DATA_BLOCK "DB_Parameters"
{ S7_Optimized_Access := 'TRUE' }
VERSION : 0.1
   VAR
      Level_Low : Real := 30.0;
      Level_High : Real := 80.0;
      Level_CritHigh : Real := 95.0;
      Source_Min : Real := 15.0;
      Source_Hyst_pct : Real := 5.0;
      Flow_Min : Real := 2.0;
      Flow_Validation : Time := T#10s;
      Restart_Delay : Time := T#30s;
      Run_Feedback_Timeout : Time := T#5s;
      Init_Delay : Time := T#2s;
      Maint_Test_Max : Time := T#60s;
      FreqStarts_Max : Int := 3;
      FreqStarts_Window_min : Int := 60;
      Current_Nominal : Real := 10.0;
      Current_High : Real := 12.0;
      Current_High_Delay : Time := T#5s;
      Maintenance_Interval_h : Real := 500.0;
      Raw_Low_Limit : Int := -500;
      Raw_High_Limit : Int := 28500;
      LevelRise_Window : Time := T#60s;
      LevelRise_Min : Real := 0.5;
      Tank_Volume : Real := 10.0;
      Pump_Flow : Real := 12.0;
      Drain_Flow : Real := 3.0;
      Sim_Step : Real := 0.1;
      Time_Accel : Real := 1.0;
   END_VAR

BEGIN

END_DATA_BLOCK